PROGRAM Intfc_Right_PK
VAR
END_VAR

// NETWORK 1

END_PROGRAM

(* stored: Version 1.1.0.1, ProductVersion 3.1.4022.11
   POU Intfc_Right_PK: Id {b0a5da56-5077-426d-abb2-f3dd5a7d9ff3}, SpecialFunc None *)
